KUKA KRL data list: PROTON_EXHIBITION.dat

&ACCESS RVP
&REL 2
&PARAM DISKPATH = KRC:\\R1\\Program
DEFDAT  PROTON_EXHIBITION
;FOLD EXTERNAL DECLARATIONS;%{PE}%MKUKATPBASIS,%CEXT,%VCOMMON,%P
;FOLD BASISTECH EXT;%{PE}%MKUKATPBASIS,%CEXT,%VEXT,%P
EXT  BAS (BAS_COMMAND  :IN,REAL  :IN )
DECL INT SUCCESS
;ENDFOLD (BASISTECH EXT)
;FOLD USER EXT;%{E}%MKUKATPUSER,%CEXT,%VEXT,%P
;Make your modifications here

;ENDFOLD (USER EXT)
;ENDFOLD (EXTERNAL DECLARATIONS)
DECL E6POS XP1={ X 72.744058, Y 1040.860681, Z 983.603439, A -160.000000, B 0.000051, C 90.000000, S 22, T 19, E1 0.0, E2 0.0, E3 0.0, E4 0.0, E5 0.0, E6 0.0 }
DECL FDAT FP1 = { BASE_NO 0, TOOL_NO 1, IPO_FRAME #BASE, POINT2[] " " }
DECL PDAT PPDAT1={ACC 100.000,APO_DIST 500.000,APO_MODE #CDIS,GEAR_JERK 100.000,EXAX_IGN 0}
DECL E6POS XP2={ X 106.398535, Y 965.069035, Z 479.071032, A -160.000018, B 0.000056, C 134.999980, S 22, T 19, E1 0.0, E2 0.0, E3 0.0, E4 0.0, E5 0.0, E6 0.0 }
DECL FDAT FP2 = { BASE_NO 0, TOOL_NO 1, IPO_FRAME #BASE, POINT2[] " " }
DECL PDAT PPDAT2={ACC 100.000,APO_DIST 500.000,APO_MODE #CDIS,GEAR_JERK 100.000,EXAX_IGN 0}
DECL E6POS XP3={ X 112.668856, Y 947.841308, Z 479.070952, A -160.000015, B 0.000050, C 119.999992, S 22, T 19, E1 0.0, E2 0.0, E3 0.0, E4 0.0, E5 0.0, E6 0.0 }
DECL FDAT FP3 = { BASE_NO 0, TOOL_NO 1, IPO_FRAME #BASE, POINT2[] " " }
DECL PDAT PPDAT3={ACC 100.000,APO_DIST 500.000,APO_MODE #CDIS,GEAR_JERK 100.000,EXAX_IGN 0}
DECL E6POS XP4={ X 112.668856, Y 947.841308, Z 479.070952, A -160.000015, B 0.000050, C 119.999992, S 22, T 19, E1 0.0, E2 0.0, E3 0.0, E4 0.0, E5 0.0, E6 0.0 }
DECL FDAT FP4 = { BASE_NO 0, TOOL_NO 1, IPO_FRAME #BASE, POINT2[] " " }
DECL PDAT PPDAT4={ACC 100.000,APO_DIST 500.000,APO_MODE #CDIS,GEAR_JERK 100.000,EXAX_IGN 0}
DECL E6POS XP5={ X 118.939200, Y 930.613562, Z 479.070894, A 19.999984, B -0.000057, C -104.999996, S 22, T 19, E1 0.0, E2 0.0, E3 0.0, E4 0.0, E5 0.0, E6 0.0 }
DECL FDAT FP5 = { BASE_NO 0, TOOL_NO 1, IPO_FRAME #BASE, POINT2[] " " }
DECL PDAT PPDAT5={ACC 100.000,APO_DIST 500.000,APO_MODE #CDIS,GEAR_JERK 100.000,EXAX_IGN 0}
DECL E6POS XP6={ X 118.939200, Y 930.613562, Z 479.070894, A 19.999984, B -0.000057, C -104.999996, S 22, T 19, E1 0.0, E2 0.0, E3 0.0, E4 0.0, E5 0.0, E6 0.0 }
DECL FDAT FP6 = { BASE_NO 0, TOOL_NO 1, IPO_FRAME #BASE, POINT2[] " " }
DECL PDAT PPDAT6={ACC 100.000,APO_DIST 500.000,APO_MODE #CDIS,GEAR_JERK 100.000,EXAX_IGN 0}
DECL E6POS XP7={ X 125.209589, Y 913.385922, Z 479.070942, A 19.999960, B -0.000044, C -90.000001, S 22, T 19, E1 0.0, E2 0.0, E3 0.0, E4 0.0, E5 0.0, E6 0.0 }
DECL FDAT FP7 = { BASE_NO 0, TOOL_NO 1, IPO_FRAME #BASE, POINT2[] " " }
DECL PDAT PPDAT7={ACC 100.000,APO_DIST 500.000,APO_MODE #CDIS,GEAR_JERK 100.000,EXAX_IGN 0}
DECL E6POS XP8={ X 125.209589, Y 913.385922, Z 479.070942, A 19.999960, B -0.000044, C -90.000001, S 22, T 19, E1 0.0, E2 0.0, E3 0.0, E4 0.0, E5 0.0, E6 0.0 }
DECL FDAT FP8 = { BASE_NO 0, TOOL_NO 1, IPO_FRAME #BASE, POINT2[] " " }
DECL PDAT PPDAT8={ACC 100.000,APO_DIST 500.000,APO_MODE #CDIS,GEAR_JERK 100.000,EXAX_IGN 0}
DECL E6POS XP9={ X 131.480033, Y 896.158220, Z 479.070968, A 19.999973, B -0.000043, C -74.999983, S 22, T 19, E1 0.0, E2 0.0, E3 0.0, E4 0.0, E5 0.0, E6 0.0 }
DECL FDAT FP9 = { BASE_NO 0, TOOL_NO 1, IPO_FRAME #BASE, POINT2[] " " }
DECL PDAT PPDAT9={ACC 100.000,APO_DIST 500.000,APO_MODE #CDIS,GEAR_JERK 100.000,EXAX_IGN 0}
DECL E6POS XP10={ X 131.480033, Y 896.158220, Z 479.070968, A 19.999973, B -0.000043, C -74.999983, S 22, T 19, E1 0.0, E2 0.0, E3 0.0, E4 0.0, E5 0.0, E6 0.0 }
DECL FDAT FP10 = { BASE_NO 0, TOOL_NO 1, IPO_FRAME #BASE, POINT2[] " " }
DECL PDAT PPDAT10={ACC 100.000,APO_DIST 500.000,APO_MODE #CDIS,GEAR_JERK 100.000,EXAX_IGN 0}
DECL E6POS XP11={ X 134.330152, Y 888.327419, Z 479.071105, A 19.999986, B -0.000028, C -59.999982, S 22, T 19, E1 0.0, E2 0.0, E3 0.0, E4 0.0, E5 0.0, E6 0.0 }
DECL FDAT FP11 = { BASE_NO 0, TOOL_NO 1, IPO_FRAME #BASE, POINT2[] " " }
DECL PDAT PPDAT11={ACC 100.000,APO_DIST 500.000,APO_MODE #CDIS,GEAR_JERK 100.000,EXAX_IGN 0}
DECL E6POS XP12={ X 134.330152, Y 888.327419, Z 479.071105, A 19.999986, B -0.000028, C -59.999982, S 22, T 19, E1 0.0, E2 0.0, E3 0.0, E4 0.0, E5 0.0, E6 0.0 }
DECL FDAT FP12 = { BASE_NO 0, TOOL_NO 1, IPO_FRAME #BASE, POINT2[] " " }
DECL PDAT PPDAT12={ACC 100.000,APO_DIST 500.000,APO_MODE #CDIS,GEAR_JERK 100.000,EXAX_IGN 0}
DECL E6POS XP13={ X 72.744058, Y 1040.860681, Z 983.603439, A -160.000000, B 0.000051, C 90.000000, S 22, T 19, E1 0.0, E2 0.0, E3 0.0, E4 0.0, E5 0.0, E6 0.0 }
DECL FDAT FP13 = { BASE_NO 0, TOOL_NO 1, IPO_FRAME #BASE, POINT2[] " " }
DECL PDAT PPDAT13={ACC 100.000,APO_DIST 500.000,APO_MODE #CDIS,GEAR_JERK 100.000,EXAX_IGN 0}
ENDDAT
